Fanuc KAREL source: IO0049.KL

-- PROVISIONAL review KL for V1013-1; original PC SHA256 fd31c3501554630f1e0b661b38b4c9af98b2351f287f29bcb595060e74b3d7f0
-- Incomplete behavior may be omitted. Consult companion uncertainty JSON. Do not deploy.
PROGRAM IO0049
%NOLOCKGROUP
-- UNRESOLVED_LOCAL_POOL 5 cells at code offset 13; source declarations unknown
-- DIRECT_LOCAL_WORD_ACCESS alone does not prove INTEGER, REAL, or BOOLEAN
BEGIN
  -- UNRESOLVED_PC offsets 0-18; opcodes 2B,2C,7B
  -- UNRESOLVED_PC offsets 23-30; opcodes 9D,23
  -- UNRESOLVED_PC offsets 35-49; opcodes 2E,22,9D,33,35
  -- UNRESOLVED_PC offsets 54-61; opcodes 9D,23
  -- UNRESOLVED_PC offsets 66-77; opcodes 2E,23
  -- UNRESOLVED_PC offsets 82-86; opcodes 9D,9D,1A
  -- UNRESOLVED_PC offsets 91-95; opcodes 7F
  -- UNRESOLVED_PC offsets 100-104; opcodes 27,AA
  -- UNRESOLVED_PC offsets 109-113; opcodes 7F
END IO0049
